// TIA Portal V17 export
// export: Created 2023-12-22T15:04:44.804435Z, ExportSetting WithDefaults, DisplayName Totally Integrated Automation Portal, DisplayVersion V17, DisplayName TIA Portal Openness, DisplayVersion V17, DisplayName TIA Portal Version Control Interface, DisplayVersion V17, DisplayName STEP 7 Professional, DisplayVersion V17, DisplayName STEP 7 Safety, DisplayVersion V17, DisplayName WinCC Advanced, DisplayVersion V17
DATA_BLOCK "ModBus_TCP_DB"   // DB40
VERSION : 0.1
// stored: AutoNumber false, DBAccessibleFromOPCUA true, InstanceOfName ModBus_TCP, InstanceOfType FB
"ModBus_TCP"
   // VAR RETAIN
   //    DATA : Array[0..100] of Word;
   //    CONNECT { S7_SetPoint := 'True'} : TCON_IP_v4;
   // END_VAR
BEGIN
   DATA[0..100] := 16#0000;
   CONNECT.InterfaceId := 64;
   CONNECT.ID := 16#0001;
   CONNECT.ConnectionType := 16#0B;
   CONNECT.ActiveEstablished := TRUE;
   CONNECT.RemoteAddress.ADDR[1] := 16#0A;
   CONNECT.RemoteAddress.ADDR[2..3] := 16#01;
   CONNECT.RemoteAddress.ADDR[4] := 16#C9;
   CONNECT.RemotePort := 503;
   CONNECT.LocalPort := 0;
END_DATA_BLOCK
